// TIA Portal V20 export
TYPE "typeCmInterfaceSoftCam"
// stored: Access Published, Namespace Unit1.Em4
   STRUCT
      positionMoving : "Unit1.Em4.typeCmInterfaceSoftCamPositionMoving";
   END_STRUCT;
END_TYPE
